RoboDK station: Example 2.1 - Pick and Place options.rdk

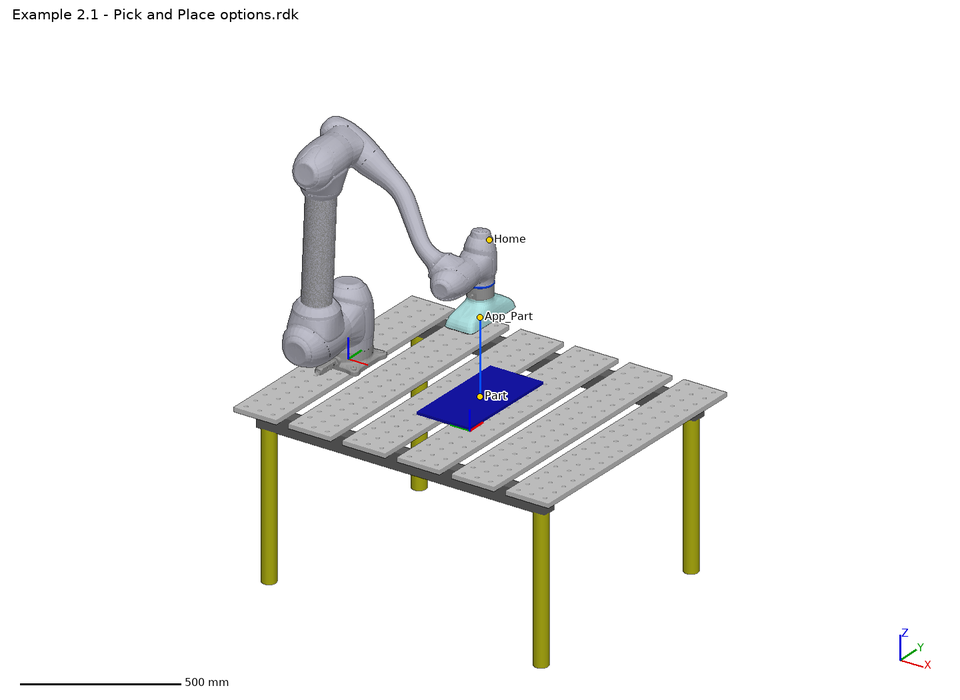
[picture v0: the station drawn from its stored meshes, robots at their saved joint values, targets as dots, program paths as lines]
Station Example 2.1 - Pick and Place options. Poses are relative to the parent item; angles as X-Y-Z fixed-axis rotations.
  - frame Doosan Robotics M1013 Base at (0, 0, 0) mm
    - robot Doosan Robotics M1013: 6 axes, payload 10 kg, reach 1300 mm, repeatability 0.1 mm, weight 33 kg
        modified DH rows (alpha deg, a mm, theta deg, d mm): 0, 0, 0, 152.5; -90, 0, -90, 34.506; 0, 620, -90, 0; -90, 0, 0, 559; 90, 0, 0, 0; -90, 0, 180, 121
        base shift (0, 0, 0) mm, rotated rx 0 ry 0 rz 180 deg
        joint limits [-360, -360, -160, -360, -360, -360] to [360, 360, 160, 360, 360, 360]; home [0, 0, -90, 0, 0, 0]; saved at [3.957, -2.294, -119.719, 0, -57.987, 3.957]
      - tool Vaccum, TCP at (0, 0, 69.67) mm, size 247.5 x 110 x 75.9 mm, geometry from Vaccum.step
  - frame World at (0, 0, 0) mm
    - target Home (joint target) at (559, -34.51, 581.83) mm, rotated rx 180 ry 0 rz 90 deg; joints [0, 0, -90, 0, -90, 0] of Doosan Robotics M1013
    - object Table at (500, 0, 0) mm, size 1193.8 x 965.2 x 609.6 mm, geometry from welding_table.sld
  - frame Part at (600, -200, 0) mm, rotated rx 0 ry 0 rz 90.06 deg
    - target Part (Cartesian target) at (200.11, 99.78, 10) mm, rotated rx 180 ry 0 rz -0.06 deg; joints [35.378, -13.73, -158.686, 0, -7.583, 125.442] of Doosan Robotics M1013
    - target App_Part (Cartesian target) at (200.11, 99.78, 285) mm, rotated rx 180 ry 0 rz -0.06 deg; joints [3.957, -2.294, -119.719, 0, -57.987, 3.957] of Doosan Robotics M1013
    - object Part at (0, 0, 0) mm, size 400 x 200 x 10 mm, geometry from Part.step
  - program PickPart (6 instructions, listed below)
  - program ReplaceObjects (1 instructions, listed below)
  - program GoHome (3 instructions, listed below)
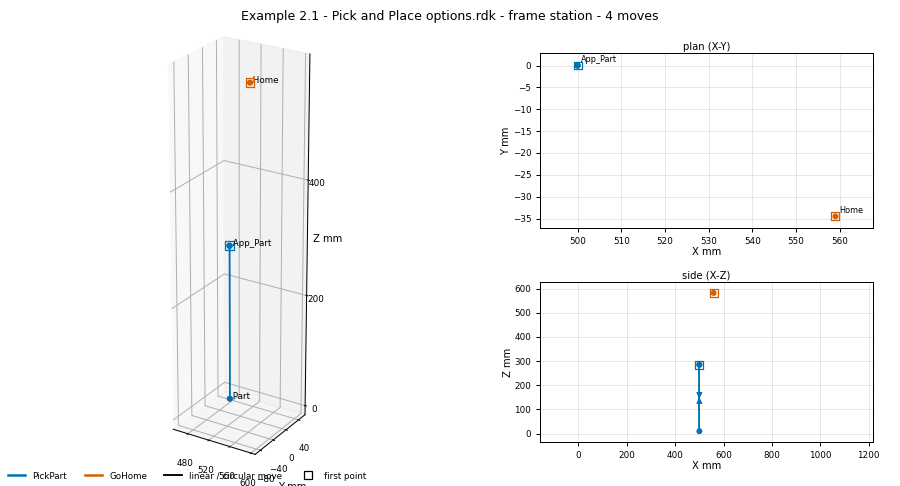
[picture p0: tool path of Example 2.1 - Pick and Place options.rdk in frame station, 4 of 4 moves have a stored position in this frame; points joined in program order, loops and branches not executed]

--- program PickPart (robot Doosan Robotics M1013) ---
  Set Ref.: Part
  Set Tool: Vaccum
  MoveJ (App_Part)
  MoveL (Part)
  Attach to Vaccum
  MoveL (App_Part)

--- program ReplaceObjects (robot Doosan Robotics M1013) ---
  Replace objects

--- program GoHome (robot Doosan Robotics M1013) ---
  Set Ref.: World
  Set Tool: Vaccum
  MoveJ (Home)
